// TIA Portal project "实验五_V20" (V20)

(* hardware
DEVICE "S7-300/ET200M station_1"  S7-300 station
   slot 0: "导轨_0"  Rail  6ES7 390-1***0-0AA0
   slot 2: "PLC_1"  CPU 314C-2 DP  6ES7 314-6CG03-0AB0  V2.6
      slot 0: "MPI 接口_1"  X1
      slot 1: "DP 接口_1"  X2
      slot 2: "DI 24/DO 16_1"  DI24/DO16
      slot 3: "AI 5/AO 2_1"  AI5/AO2
      slot 4: "计数_1"  Counter
      slot 5: "定位_1"  Positioning
*)

// ===== PLC "PLC_1"  CPU 314C-2 DP =====

VAR_GLOBAL   // PLC tag table "默认变量表"
   "Tag_1" AT %M1.1 : Bool;
END_VAR

VAR_GLOBAL   // PLC tag table "变量表_1"
   "四层内选按钮" AT %I0.0 : Bool;
   "三层内选按钮" AT %I0.1 : Bool;
   "二层内选按钮" AT %I0.2 : Bool;
   "一层内选按钮" AT %I0.3 : Bool;
   "四层下呼按钮" AT %I0.4 : Bool;
   "三层下呼按钮" AT %I0.5 : Bool;
   "二层下呼按钮" AT %I0.6 : Bool;
   "一层上呼按钮" AT %I0.7 : Bool;
   "二层上呼按钮" AT %I1.0 : Bool;
   "三层上呼按钮" AT %I1.1 : Bool;
   "一层行程开关" AT %I1.2 : Bool;
   "二层行程开关" AT %I1.3 : Bool;
   "三层行程开关" AT %I1.4 : Bool;
   "四层行程开关" AT %I1.5 : Bool;
   "四层指示" AT %Q4.0 : Bool;
   "三层指示" AT %Q4.1 : Bool;
   "二层指示" AT %Q4.2 : Bool;
   "一层指示" AT %Q4.3 : Bool;
   "轿厢下降指示" AT %Q4.4 : Bool;
   "轿厢上升指示" AT %Q4.5 : Bool;
   "四层内选指示" AT %Q4.6 : Bool;
   "三层内选指示" AT %Q4.7 : Bool;
   "二层内选指示" AT %Q5.0 : Bool;
   "一层内选指示" AT %Q5.1 : Bool;
   "一层上呼指示" AT %Q5.2 : Bool;
   "二层上呼指示" AT %Q5.3 : Bool;
   "三层上呼指示" AT %Q5.4 : Bool;
   "二层下呼指示" AT %Q5.5 : Bool;
   "三层下呼指示" AT %Q5.6 : Bool;
   "四层下呼指示" AT %Q5.7 : Bool;
   "1上" AT %M10.0 : Bool;
   "2上" AT %M10.1 : Bool;
   "3上" AT %M10.2 : Bool;
   "2下" AT %M10.3 : Bool;
   "3下" AT %M10.4 : Bool;
   "4下" AT %M10.5 : Bool;
   "电梯一层登记" AT %M10.6 : Bool;
   "电梯二层登记" AT %M10.7 : Bool;
   "电梯三层登记" AT %M11.0 : Bool;
   "电梯四层登记" AT %M11.1 : Bool;
   "中继11" AT %M11.2 : Bool;
   "中继12" AT %M11.3 : Bool;
   "中继13" AT %M11.4 : Bool;
   "中继14" AT %M11.5 : Bool;
   "中继15" AT %M11.6 : Bool;
   "中继16" AT %M11.7 : Bool;
   "中继17" AT %M12.0 : Bool;
   "中继18" AT %M12.1 : Bool;
END_VAR

DATA_BLOCK "数据块_1"   // DB1
{ S7_Optimized_Access := 'FALSE' }
VERSION : 0.1
   VAR
      当前楼层数 : Int;
   END_VAR
BEGIN
END_DATA_BLOCK

FUNCTION "行程开关" : Void   // FC1, LAD
{ S7_Optimized_Access := 'FALSE' }
VERSION : 0.1
BEGIN

REGION Network 1
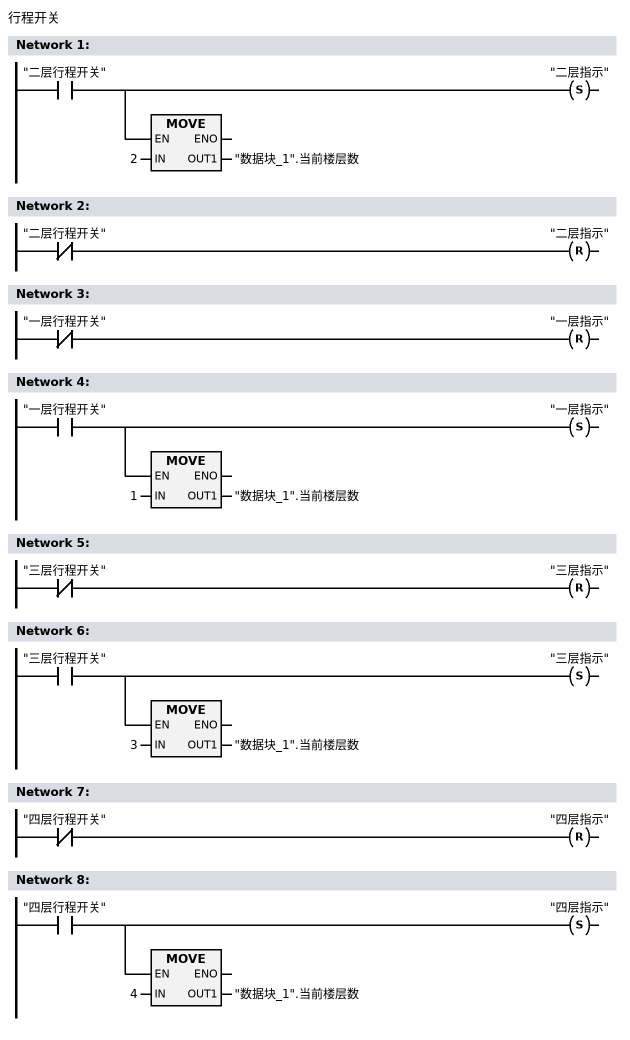
   RUNG wire#powerrail
      Contact( "二层行程开关" )
      wire#w1
      S_Coil( "二层指示" )
   END_RUNG
   RUNG wire#w1
      { S7_GenerateENO := "TRUE" } Move(in := 2, out1 => "数据块_1".当前楼层数)
   END_RUNG
   // the same network as SCL:
   IF "二层行程开关" THEN
       "二层指示" := TRUE;
       "数据块_1".当前楼层数 := 2;
   END_IF;
END_REGION

REGION Network 2
   RUNG wire#powerrail
      I_Contact( "二层行程开关" )
      R_Coil( "二层指示" )
   END_RUNG
   // the same network as SCL:
   IF NOT "二层行程开关" THEN "二层指示" := FALSE; END_IF;
END_REGION

REGION Network 3
   RUNG wire#powerrail
      I_Contact( "一层行程开关" )
      R_Coil( "一层指示" )
   END_RUNG
   // the same network as SCL:
   IF NOT "一层行程开关" THEN "一层指示" := FALSE; END_IF;
END_REGION

REGION Network 4
   RUNG wire#powerrail
      Contact( "一层行程开关" )
      wire#w1
      S_Coil( "一层指示" )
   END_RUNG
   RUNG wire#w1
      { S7_GenerateENO := "TRUE" } Move(in := 1, out1 => "数据块_1".当前楼层数)
   END_RUNG
   // the same network as SCL:
   IF "一层行程开关" THEN
       "一层指示" := TRUE;
       "数据块_1".当前楼层数 := 1;
   END_IF;
END_REGION

REGION Network 5
   RUNG wire#powerrail
      I_Contact( "三层行程开关" )
      R_Coil( "三层指示" )
   END_RUNG
   // the same network as SCL:
   IF NOT "三层行程开关" THEN "三层指示" := FALSE; END_IF;
END_REGION

REGION Network 6
   RUNG wire#powerrail
      Contact( "三层行程开关" )
      wire#w1
      S_Coil( "三层指示" )
   END_RUNG
   RUNG wire#w1
      { S7_GenerateENO := "TRUE" } Move(in := 3, out1 => "数据块_1".当前楼层数)
   END_RUNG
   // the same network as SCL:
   IF "三层行程开关" THEN
       "三层指示" := TRUE;
       "数据块_1".当前楼层数 := 3;
   END_IF;
END_REGION

REGION Network 7
   RUNG wire#powerrail
      I_Contact( "四层行程开关" )
      R_Coil( "四层指示" )
   END_RUNG
   // the same network as SCL:
   IF NOT "四层行程开关" THEN "四层指示" := FALSE; END_IF;
END_REGION

REGION Network 8
   RUNG wire#powerrail
      Contact( "四层行程开关" )
      wire#w1
      S_Coil( "四层指示" )
   END_RUNG
   RUNG wire#w1
      { S7_GenerateENO := "TRUE" } Move(in := 4, out1 => "数据块_1".当前楼层数)
   END_RUNG
   // the same network as SCL:
   IF "四层行程开关" THEN
       "四层指示" := TRUE;
       "数据块_1".当前楼层数 := 4;
   END_IF;
END_REGION
END_FUNCTION

FUNCTION "桥内面" : Void   // FC2, LAD
{ S7_Optimized_Access := 'FALSE' }
VERSION : 0.1
BEGIN

REGION Network 1
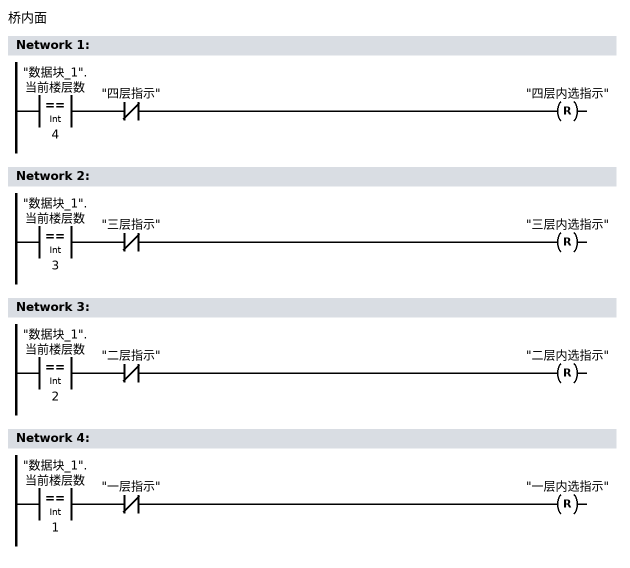
   RUNG wire#powerrail
      { S7_Templates := "SrcType := Int" } EQ_Contact(in1 := "数据块_1".当前楼层数, in2 := 4)
      I_Contact( "四层指示" )
      R_Coil( "四层内选指示" )
   END_RUNG
   // the same network as SCL:
   IF ("数据块_1".当前楼层数 = 4) AND NOT "四层指示" THEN "四层内选指示" := FALSE; END_IF;
END_REGION

REGION Network 2
   RUNG wire#powerrail
      { S7_Templates := "SrcType := Int" } EQ_Contact(in1 := "数据块_1".当前楼层数, in2 := 3)
      I_Contact( "三层指示" )
      R_Coil( "三层内选指示" )
   END_RUNG
   // the same network as SCL:
   IF ("数据块_1".当前楼层数 = 3) AND NOT "三层指示" THEN "三层内选指示" := FALSE; END_IF;
END_REGION

REGION Network 3
   RUNG wire#powerrail
      { S7_Templates := "SrcType := Int" } EQ_Contact(in1 := "数据块_1".当前楼层数, in2 := 2)
      I_Contact( "二层指示" )
      R_Coil( "二层内选指示" )
   END_RUNG
   // the same network as SCL:
   IF ("数据块_1".当前楼层数 = 2) AND NOT "二层指示" THEN "二层内选指示" := FALSE; END_IF;
END_REGION

REGION Network 4
   RUNG wire#powerrail
      { S7_Templates := "SrcType := Int" } EQ_Contact(in1 := "数据块_1".当前楼层数, in2 := 1)
      I_Contact( "一层指示" )
      R_Coil( "一层内选指示" )
   END_RUNG
   // the same network as SCL:
   IF ("数据块_1".当前楼层数 = 1) AND NOT "一层指示" THEN "一层内选指示" := FALSE; END_IF;
END_REGION
END_FUNCTION

FUNCTION "楼层登记" : Void   // FC3, LAD
{ S7_Optimized_Access := 'FALSE' }
VERSION : 0.1
BEGIN

REGION Network 1
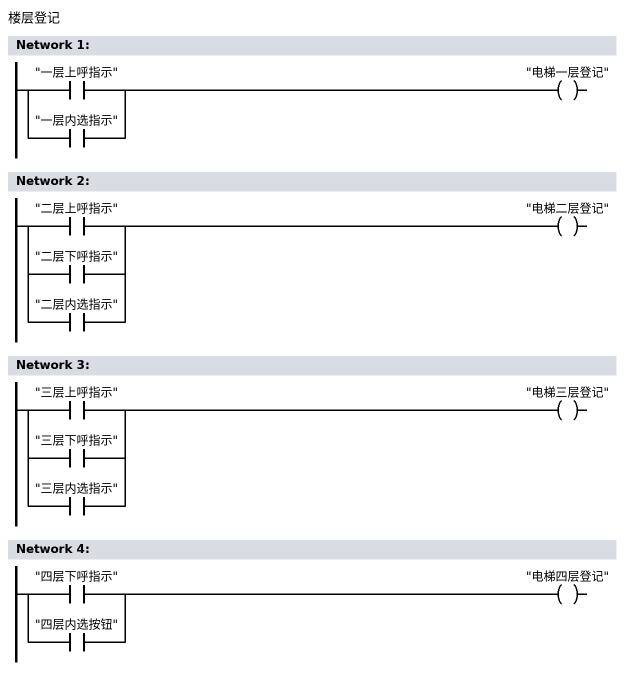
   RUNG wire#powerrail
      Contact( "一层上呼指示" )
      wire#w1
      Coil( "电梯一层登记" )
   END_RUNG
   RUNG wire#powerrail
      Contact( "一层内选指示" )
   END_RUNG wire#w1
   // the same network as SCL:
   "电梯一层登记" := "一层上呼指示" OR "一层内选指示";
END_REGION

REGION Network 2
   RUNG wire#powerrail
      Contact( "二层上呼指示" )
      wire#w1
      Coil( "电梯二层登记" )
   END_RUNG
   RUNG wire#powerrail
      Contact( "二层下呼指示" )
   END_RUNG wire#w1
   RUNG wire#powerrail
      Contact( "二层内选指示" )
   END_RUNG wire#w1
   // the same network as SCL:
   "电梯二层登记" := "二层上呼指示" OR "二层下呼指示" OR "二层内选指示";
END_REGION

REGION Network 3
   RUNG wire#powerrail
      Contact( "三层上呼指示" )
      wire#w1
      Coil( "电梯三层登记" )
   END_RUNG
   RUNG wire#powerrail
      Contact( "三层下呼指示" )
   END_RUNG wire#w1
   RUNG wire#powerrail
      Contact( "三层内选指示" )
   END_RUNG wire#w1
   // the same network as SCL:
   "电梯三层登记" := "三层上呼指示" OR "三层下呼指示" OR "三层内选指示";
END_REGION

REGION Network 4
   RUNG wire#powerrail
      Contact( "四层下呼指示" )
      wire#w1
      Coil( "电梯四层登记" )
   END_RUNG
   RUNG wire#powerrail
      Contact( "四层内选按钮" )
   END_RUNG wire#w1
   // the same network as SCL:
   "电梯四层登记" := "四层下呼指示" OR "四层内选按钮";
END_REGION
END_FUNCTION

FUNCTION "内选灯控制" : Void   // FC4, LAD
{ S7_Optimized_Access := 'FALSE' }
VERSION : 0.1
BEGIN

REGION Network 1
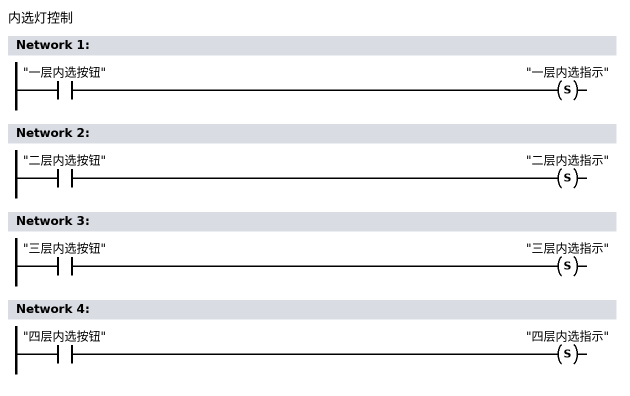
   RUNG wire#powerrail
      Contact( "一层内选按钮" )
      S_Coil( "一层内选指示" )
   END_RUNG
   // the same network as SCL:
   IF "一层内选按钮" THEN "一层内选指示" := TRUE; END_IF;
END_REGION

REGION Network 2
   RUNG wire#powerrail
      Contact( "二层内选按钮" )
      S_Coil( "二层内选指示" )
   END_RUNG
   // the same network as SCL:
   IF "二层内选按钮" THEN "二层内选指示" := TRUE; END_IF;
END_REGION

REGION Network 3
   RUNG wire#powerrail
      Contact( "三层内选按钮" )
      S_Coil( "三层内选指示" )
   END_RUNG
   // the same network as SCL:
   IF "三层内选按钮" THEN "三层内选指示" := TRUE; END_IF;
END_REGION

REGION Network 4
   RUNG wire#powerrail
      Contact( "四层内选按钮" )
      S_Coil( "四层内选指示" )
   END_RUNG
   // the same network as SCL:
   IF "四层内选按钮" THEN "四层内选指示" := TRUE; END_IF;
END_REGION
END_FUNCTION

FUNCTION "外呼" : Void   // FC5, LAD
{ S7_Optimized_Access := 'FALSE' }
VERSION : 0.1
BEGIN

REGION Network 1
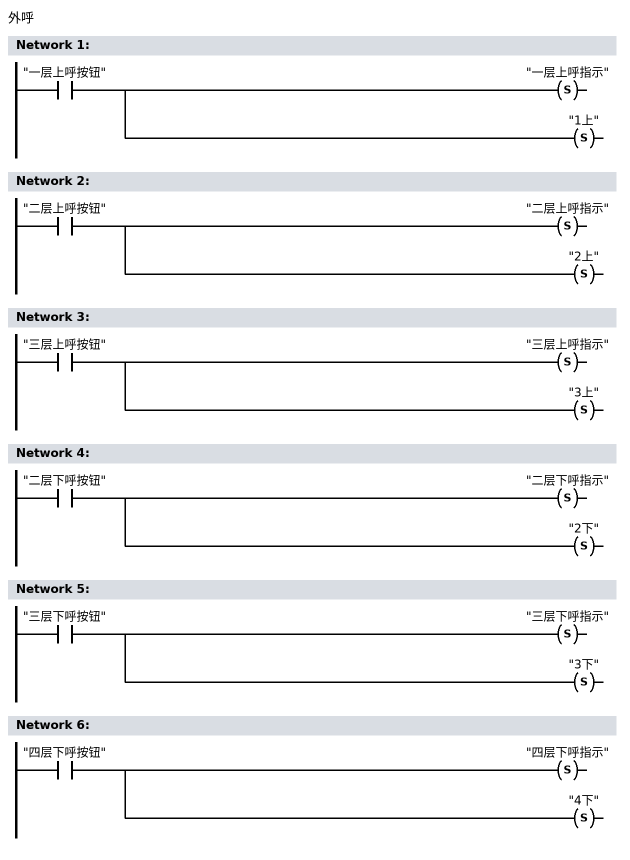
   RUNG wire#powerrail
      Contact( "一层上呼按钮" )
      wire#w1
      S_Coil( "一层上呼指示" )
   END_RUNG
   RUNG wire#w1
      S_Coil( "1上" )
   END_RUNG
   // the same network as SCL:
   IF "一层上呼按钮" THEN
       "一层上呼指示" := TRUE;
       "1上" := TRUE;
   END_IF;
END_REGION

REGION Network 2
   RUNG wire#powerrail
      Contact( "二层上呼按钮" )
      wire#w1
      S_Coil( "二层上呼指示" )
   END_RUNG
   RUNG wire#w1
      S_Coil( "2上" )
   END_RUNG
   // the same network as SCL:
   IF "二层上呼按钮" THEN
       "二层上呼指示" := TRUE;
       "2上" := TRUE;
   END_IF;
END_REGION

REGION Network 3
   RUNG wire#powerrail
      Contact( "三层上呼按钮" )
      wire#w1
      S_Coil( "三层上呼指示" )
   END_RUNG
   RUNG wire#w1
      S_Coil( "3上" )
   END_RUNG
   // the same network as SCL:
   IF "三层上呼按钮" THEN
       "三层上呼指示" := TRUE;
       "3上" := TRUE;
   END_IF;
END_REGION

REGION Network 4
   RUNG wire#powerrail
      Contact( "二层下呼按钮" )
      wire#w1
      S_Coil( "二层下呼指示" )
   END_RUNG
   RUNG wire#w1
      S_Coil( "2下" )
   END_RUNG
   // the same network as SCL:
   IF "二层下呼按钮" THEN
       "二层下呼指示" := TRUE;
       "2下" := TRUE;
   END_IF;
END_REGION

REGION Network 5
   RUNG wire#powerrail
      Contact( "三层下呼按钮" )
      wire#w1
      S_Coil( "三层下呼指示" )
   END_RUNG
   RUNG wire#w1
      S_Coil( "3下" )
   END_RUNG
   // the same network as SCL:
   IF "三层下呼按钮" THEN
       "三层下呼指示" := TRUE;
       "3下" := TRUE;
   END_IF;
END_REGION

REGION Network 6
   RUNG wire#powerrail
      Contact( "四层下呼按钮" )
      wire#w1
      S_Coil( "四层下呼指示" )
   END_RUNG
   RUNG wire#w1
      S_Coil( "4下" )
   END_RUNG
   // the same network as SCL:
   IF "四层下呼按钮" THEN
       "四层下呼指示" := TRUE;
       "4下" := TRUE;
   END_IF;
END_REGION
END_FUNCTION

FUNCTION "外呼灭" : Void   // FC6, LAD
{ S7_Optimized_Access := 'FALSE' }
VERSION : 0.1
BEGIN

REGION Network 1
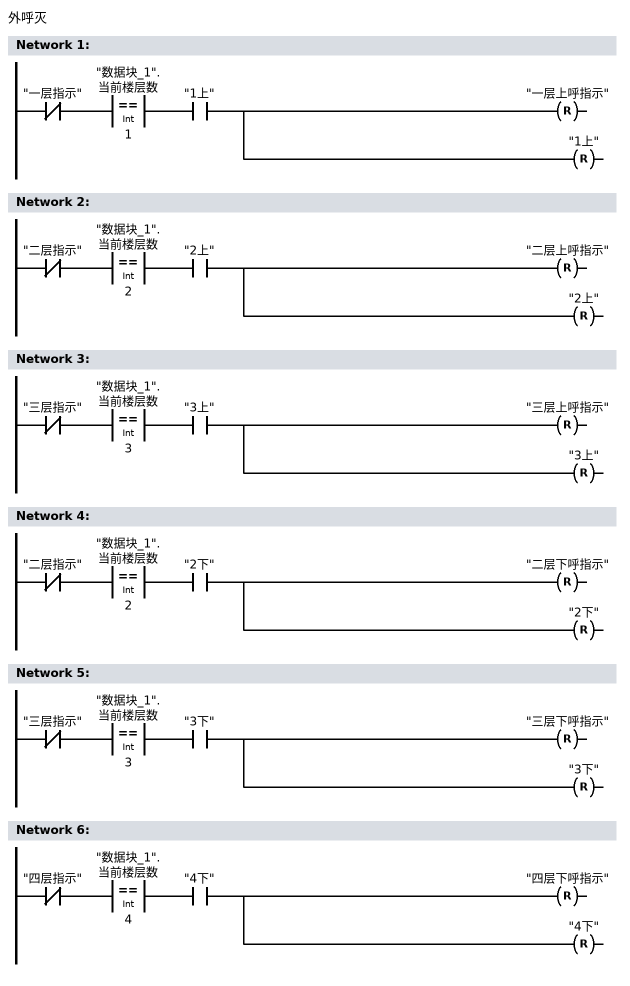
   RUNG wire#powerrail
      I_Contact( "一层指示" )
      { S7_Templates := "SrcType := Int" } EQ_Contact(in1 := "数据块_1".当前楼层数, in2 := 1)
      Contact( "1上" )
      wire#w1
      R_Coil( "一层上呼指示" )
   END_RUNG
   RUNG wire#w1
      R_Coil( "1上" )
   END_RUNG
   // the same network as SCL:
   IF NOT "一层指示" AND ("数据块_1".当前楼层数 = 1) AND "1上" THEN
       "一层上呼指示" := FALSE;
       "1上" := FALSE;
   END_IF;
END_REGION

REGION Network 2
   RUNG wire#powerrail
      I_Contact( "二层指示" )
      { S7_Templates := "SrcType := Int" } EQ_Contact(in1 := "数据块_1".当前楼层数, in2 := 2)
      Contact( "2上" )
      wire#w1
      R_Coil( "二层上呼指示" )
   END_RUNG
   RUNG wire#w1
      R_Coil( "2上" )
   END_RUNG
   // the same network as SCL:
   IF NOT "二层指示" AND ("数据块_1".当前楼层数 = 2) AND "2上" THEN
       "二层上呼指示" := FALSE;
       "2上" := FALSE;
   END_IF;
END_REGION

REGION Network 3
   RUNG wire#powerrail
      I_Contact( "三层指示" )
      { S7_Templates := "SrcType := Int" } EQ_Contact(in1 := "数据块_1".当前楼层数, in2 := 3)
      Contact( "3上" )
      wire#w1
      R_Coil( "三层上呼指示" )
   END_RUNG
   RUNG wire#w1
      R_Coil( "3上" )
   END_RUNG
   // the same network as SCL:
   IF NOT "三层指示" AND ("数据块_1".当前楼层数 = 3) AND "3上" THEN
       "三层上呼指示" := FALSE;
       "3上" := FALSE;
   END_IF;
END_REGION

REGION Network 4
   RUNG wire#powerrail
      I_Contact( "二层指示" )
      { S7_Templates := "SrcType := Int" } EQ_Contact(in1 := "数据块_1".当前楼层数, in2 := 2)
      Contact( "2下" )
      wire#w1
      R_Coil( "二层下呼指示" )
   END_RUNG
   RUNG wire#w1
      R_Coil( "2下" )
   END_RUNG
   // the same network as SCL:
   IF NOT "二层指示" AND ("数据块_1".当前楼层数 = 2) AND "2下" THEN
       "二层下呼指示" := FALSE;
       "2下" := FALSE;
   END_IF;
END_REGION

REGION Network 5
   RUNG wire#powerrail
      I_Contact( "三层指示" )
      { S7_Templates := "SrcType := Int" } EQ_Contact(in1 := "数据块_1".当前楼层数, in2 := 3)
      Contact( "3下" )
      wire#w1
      R_Coil( "三层下呼指示" )
   END_RUNG
   RUNG wire#w1
      R_Coil( "3下" )
   END_RUNG
   // the same network as SCL:
   IF NOT "三层指示" AND ("数据块_1".当前楼层数 = 3) AND "3下" THEN
       "三层下呼指示" := FALSE;
       "3下" := FALSE;
   END_IF;
END_REGION

REGION Network 6
   RUNG wire#powerrail
      I_Contact( "四层指示" )
      { S7_Templates := "SrcType := Int" } EQ_Contact(in1 := "数据块_1".当前楼层数, in2 := 4)
      Contact( "4下" )
      wire#w1
      R_Coil( "四层下呼指示" )
   END_RUNG
   RUNG wire#w1
      R_Coil( "4下" )
   END_RUNG
   // the same network as SCL:
   IF NOT "四层指示" AND ("数据块_1".当前楼层数 = 4) AND "4下" THEN
       "四层下呼指示" := FALSE;
       "4下" := FALSE;
   END_IF;
END_REGION
END_FUNCTION

FUNCTION "选向" : Void   // FC7, LAD
{ S7_Optimized_Access := 'FALSE' }
VERSION : 0.1
BEGIN

REGION Network 1
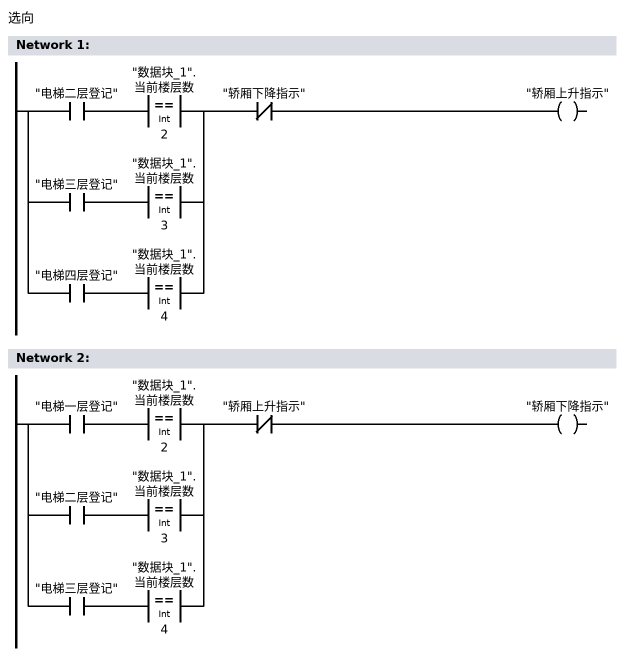
   RUNG wire#powerrail
      Contact( "电梯二层登记" )
      { S7_Templates := "SrcType := Int" } EQ_Contact(in1 := "数据块_1".当前楼层数, in2 := 2)
      wire#w1
      I_Contact( "轿厢下降指示" )
      Coil( "轿厢上升指示" )
   END_RUNG
   RUNG wire#powerrail
      Contact( "电梯三层登记" )
      { S7_Templates := "SrcType := Int" } EQ_Contact(in1 := "数据块_1".当前楼层数, in2 := 3)
   END_RUNG wire#w1
   RUNG wire#powerrail
      Contact( "电梯四层登记" )
      { S7_Templates := "SrcType := Int" } EQ_Contact(in1 := "数据块_1".当前楼层数, in2 := 4)
   END_RUNG wire#w1
   // the same network as SCL:
   "轿厢上升指示" := (("电梯二层登记" AND ("数据块_1".当前楼层数 = 2)) OR ("电梯三层登记" AND ("数据块_1".当前楼层数 = 3)) OR ("电梯四层登记" AND ("数据块_1".当前楼层数 = 4))) AND NOT "轿厢下降指示";
END_REGION

REGION Network 2
   RUNG wire#powerrail
      Contact( "电梯一层登记" )
      { S7_Templates := "SrcType := Int" } EQ_Contact(in1 := "数据块_1".当前楼层数, in2 := 2)
      wire#w1
      I_Contact( "轿厢上升指示" )
      Coil( "轿厢下降指示" )
   END_RUNG
   RUNG wire#powerrail
      Contact( "电梯二层登记" )
      { S7_Templates := "SrcType := Int" } EQ_Contact(in1 := "数据块_1".当前楼层数, in2 := 3)
   END_RUNG wire#w1
   RUNG wire#powerrail
      Contact( "电梯三层登记" )
      { S7_Templates := "SrcType := Int" } EQ_Contact(in1 := "数据块_1".当前楼层数, in2 := 4)
   END_RUNG wire#w1
   // the same network as SCL:
   "轿厢下降指示" := (("电梯一层登记" AND ("数据块_1".当前楼层数 = 2)) OR ("电梯二层登记" AND ("数据块_1".当前楼层数 = 3)) OR ("电梯三层登记" AND ("数据块_1".当前楼层数 = 4))) AND NOT "轿厢上升指示";
END_REGION
END_FUNCTION

ORGANIZATION_BLOCK "Main"   // OB1, LAD
TITLE = "Main Program Sweep (Cycle)"
{ S7_Optimized_Access := 'FALSE' }
VERSION : 0.1
   VAR_TEMP
      OB1_EV_CLASS : Byte;   // Bits 0-3 = 1 (Coming event), Bits 4-7 = 1 (Event class 1)
      OB1_SCAN_1 : Byte;   // 1 (Cold restart scan 1 of OB 1), 3 (Scan 2-n of OB 1)
      OB1_PRIORITY : Byte;   // Priority of OB Execution
      OB1_OB_NUMBR : Byte;   // 1 (Organization block 1, OB1)
      OB1_RESERVED_1 : Byte;   // Reserved for system
      OB1_RESERVED_2 : Byte;   // Reserved for system
      OB1_PREV_CYCLE : Int;   // Cycle time of previous OB1 scan (milliseconds)
      OB1_MIN_CYCLE : Int;   // Minimum cycle time of OB1 (milliseconds)
      OB1_MAX_CYCLE : Int;   // Maximum cycle time of OB1 (milliseconds)
      OB1_DATE_TIME : Date_And_Time;   // Date and time OB1 started
   END_VAR
BEGIN

REGION Network 1
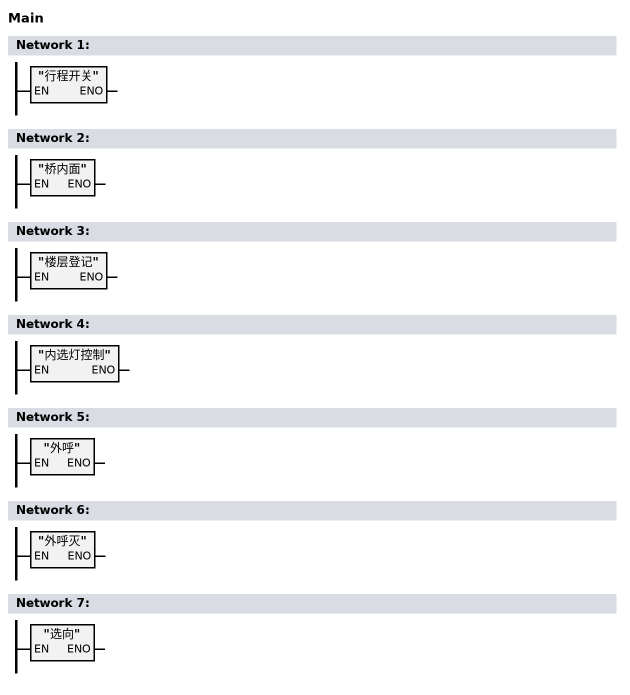
   RUNG wire#powerrail
      "行程开关"()
   END_RUNG
   // the same network as SCL:
   "行程开关"();
END_REGION

REGION Network 2
   RUNG wire#powerrail
      "桥内面"()
   END_RUNG
   // the same network as SCL:
   "桥内面"();
END_REGION

REGION Network 3
   RUNG wire#powerrail
      "楼层登记"()
   END_RUNG
   // the same network as SCL:
   "楼层登记"();
END_REGION

REGION Network 4
   RUNG wire#powerrail
      "内选灯控制"()
   END_RUNG
   // the same network as SCL:
   "内选灯控制"();
END_REGION

REGION Network 5
   RUNG wire#powerrail
      "外呼"()
   END_RUNG
   // the same network as SCL:
   "外呼"();
END_REGION

REGION Network 6
   RUNG wire#powerrail
      "外呼灭"()
   END_RUNG
   // the same network as SCL:
   "外呼灭"();
END_REGION

REGION Network 7
   RUNG wire#powerrail
      "选向"()
   END_RUNG
   // the same network as SCL:
   "选向"();
END_REGION
END_ORGANIZATION_BLOCK